{attribute 'GeneratedUsingTerminal: ATH2000-0250-0022'}
{attribute addProperty BoxType "ATH2000-0250-0022"}
{attribute addProperty Id "A_0014_ATH2050_5501_0022ATH2050_6EC099B714"}
{attribute addProperty CRC "806166480"}
{attribute addProperty Size "14"}
TYPE A_0001_ATH2000_0250_0022_300D1FD0 EXTENDS ATH2000_A7FEA1CF :
STRUCT
	{attribute addProperty Name "A_0014_ATH2050_5501_0022"}
	{attribute addProperty PreviousPort "A_0001(ATH2000-0250-0022) : B"}
	A_0014_ATH2050_5501_0022 : ATH2050_6EC099B7;
END_STRUCT
END_TYPE

(* stored: Version 1.2.0.0, ProductVersion 3.1.4024.9
   DUT A_0001_ATH2000_0250_0022_300D1FD0: Id {d24ba7d1-9afb-43d2-be42-3cd298c62340} *)
